FUNCTION_BLOCK UT_AuxiliaryOutputMapping_Type_02_Bool_NonLatched (* Type 2 Bool_NonLatched Two-position switch - returns to off *)
  (* Standard: ISO 11783-6; Classification: AUX – ISO 11783-6; Function: All Inputs; Type: UT according to ISO 11783-6; Description: Copyright (c) 2018, 2023 Jose Cabral, HR Agrartechnik GmbH This program and the accompanying materials are made available under the terms of the Eclipse Public License 2.0 which is available at https://www.eclipse.org/legal/epl-2.0/ SPDX-License-Identifier: EPL-2.0 - Type 2 Bool_NonLatched Two-position switch - returns to off Applicable to  AUX-N this maps to QX *)
  (* Version 1.0, 2018-12-05, Jose Cabral *)
  (* Version 1.1, 2022-08-04, Franz Höpfinger, HR Agrartechnik GmbH *)
  (* Version 1.2, 2023-01-05, Franz Höpfinger, HR Agrartechnik GmbH *)
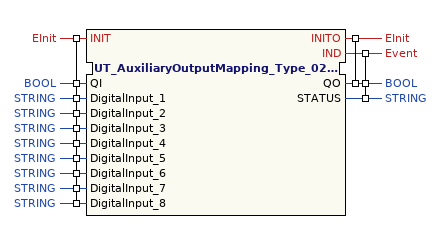
  EVENT_INPUT
    INIT : EInit WITH QI, DigitalInput_1, DigitalInput_2, DigitalInput_3, DigitalInput_4, DigitalInput_5, DigitalInput_6, DigitalInput_7, DigitalInput_8; (* Service Initialization *)
  END_EVENT
  EVENT_OUTPUT
    INITO : EInit WITH QO; (* Initialization Confirm *)
    IND WITH QO, STATUS; (* Indication from Resource *)
  END_EVENT
  VAR_INPUT
    QI : BOOL; (* Event Input Qualifier *)
    DigitalInput_1 : STRING; (* Identifier for Input 1 *)
    DigitalInput_2 : STRING; (* Identifier for Input 2 *)
    DigitalInput_3 : STRING; (* Identifier for Input 3 *)
    DigitalInput_4 : STRING; (* Identifier for Input 4 *)
    DigitalInput_5 : STRING; (* Identifier for Input 5 *)
    DigitalInput_6 : STRING; (* Identifier for Input 6 *)
    DigitalInput_7 : STRING; (* Identifier for Input 7 *)
    DigitalInput_8 : STRING; (* Identifier for Input 8 *)
  END_VAR
  VAR_OUTPUT
    QO : BOOL; (* Event Output Qualifier *)
    STATUS : STRING; (* Service Status *)
  END_VAR
END_FUNCTION_BLOCK
